(* LS Electric XG5000 project: TIME MOVE *)
(* PLC LSPLC *)
(* module base 0 slot 0: 입력 모듈:XGI-D22A/B (DC 24V 입력, 16점 (전류소스 싱크공용/ 전류소스 입력)) *)
(* module base 0 slot 1: 입력 모듈:XGI-D22A/B (DC 24V 입력, 16점 (전류소스 싱크공용/ 전류소스 입력)) *)
(* module base 0 slot 2: 출력 모듈:XGQ-RY2A/B (릴레이 출력, 16점 (2A용, Varistor 없음/Varistor 부착)) *)
(* module base 0 slot 3: 출력 모듈:XGQ-RY2A/B (릴레이 출력, 16점 (2A용, Varistor 없음/Varistor 부착)) *)

PROGRAM NewProgram (* task: 스캔 프로그램 *)
VAR
    D1 : TIME;
    P0 : BOOL;
    T1 : TON;
    이순신 : BOOL;
END_VAR

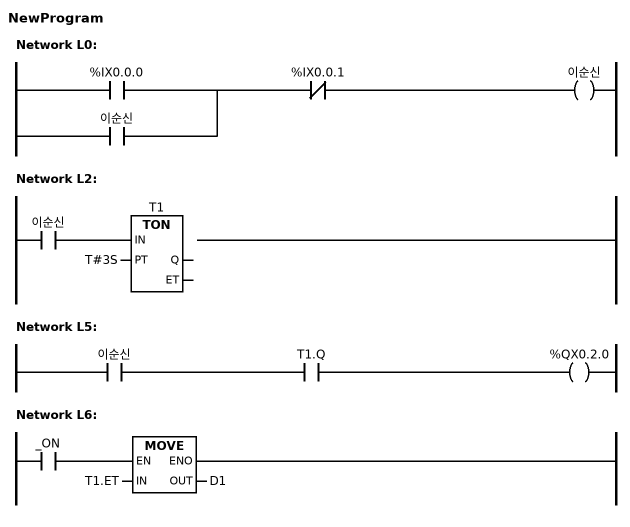
(* Rung L0 *)
이순신 := (%IX0.0.0 OR 이순신) AND NOT %IX0.0.1;
(* Rung L2 *)
T1(IN := 이순신, PT := T#3S);
(* Rung L5 *)
%QX0.2.0 := 이순신 AND T1.Q;
(* Rung L6 *)
IF _ON THEN D1 := T1.ET; END_IF;
END_PROGRAM